// TIA Portal V20 export
TYPE "typeCalibrationData"
// stored: Access Published
   STRUCT
      Align_QRCode { ExternalWritable := 'False'} : String;
      MainPNP_AxisY_Position { ExternalWritable := 'False'} : LReal;
      Align_AxisY01_POsition { ExternalWritable := 'False'} : LReal;
      Align_AxisY02_Position { ExternalWritable := 'False'} : LReal;
      Align_AxisX01_Position { ExternalWritable := 'False'} : LReal;
      Stack_Vision_data : String;
   END_STRUCT;
END_TYPE
